Universal Robots PolyScope program: HeatPWF.urp

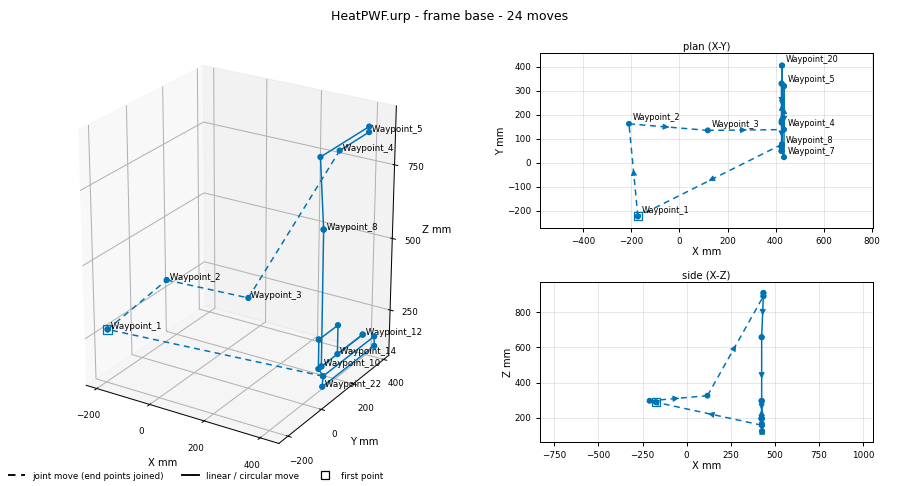
[picture p0: tool path of HeatPWF.urp in frame base, 24 of 24 moves have a stored position in this frame; points joined in program order, loops and branches not executed]
Program TDaiHeatPWF1 (installation=default directory=/programs/usbdisk_0/UR_URPs createdIn=5.11.0.108249 lastSavedIn=5.11.0.108249 robotSerialNumber=20215590035)
Calibrated DH parameters: a=[0.00016, -0.349388, -0.392209, -0.000059, 0.000026, 0]; d=[0.162575, -215.770964, 216.209801, -0.305241, 0.099656, 0.099253]; alpha=[1.570834, -0.001122, 0.007322, 1.56929, -1.570073, 0]; deltaTheta=[0, 0.606034, 5.685341, -0.008192, 0.000001, 0]
Robot Program (runOnlyOnce=true)
  MoveJ speed 60 deg/s, acceleration 80 deg/s^2 (useActiveTCP=true) feature=Base
    Waypoint Waypoint_1: TCP in base x=-173.333 y=-223.371 z=288.487 mm, rx=-2.2066 ry=-2.2292 rz=0.0202 rad; joints [-99.337, -57.321, -138.717, -73.565, 89.803, 80.13] deg; TCP offset x=0 y=0 z=26 mm, rx=0 ry=0 rz=0 rad
  MoveJ speed 60 deg/s, acceleration 80 deg/s^2 (useActiveTCP=true) feature=Base
    Waypoint Waypoint_2: TCP in base x=-210.394 y=161.858 z=296.687 mm, rx=-3.1305 ry=-0.0742 rz=0.0332 rad; joints [-187.188, -52.739, -139.358, -76.659, 90.078, 80.121] deg
  MoveJ speed 60 deg/s, acceleration 80 deg/s^2 (useActiveTCP=true) feature=Base
    Waypoint Waypoint_3: TCP in base x=117.831 y=134.656 z=325.784 mm, rx=-3.1162 ry=-0.0095 rz=0.0014 rad; joints [-262.681, -29.685, -139.379, -99.527, 90.347, 6.803] deg
  URCap Gripper Activate (Robotiq_Grippers, Robotiq Inc.) dataModel(ResetAndActivateKey=false)
  URCap Gripper (Robotiq_Grippers, Robotiq Inc.) dataModel(position=0.0, force=99.6078431372549, speed=99.6078431372549, positionInDouble=0.0, forceInDouble=99.6078431372549, speedInDouble=99.6078431372549, slaveIds=[9], blocking=true)
  MoveJ speed 60 deg/s, acceleration 80 deg/s^2 (useActiveTCP=true) feature=Base
    Waypoint Waypoint_4: TCP in base x=435.252 y=137.856 z=890.1 mm, rx=-1.5865 ry=-0.0166 rz=0.0088 rad; joints [-340.703, -101.32, -45.922, -34.906, 161.789, -2.225] deg; TCP offset x=0 y=0 z=26 mm, rx=0 ry=0 rz=0 rad
  MoveL speed 250 mm/s, acceleration 1200 mm/s^2 (useActiveTCP=true) feature=Base
    Waypoint Waypoint_5: TCP in base x=435.245 y=318.777 z=890.1 mm, rx=-1.5865 ry=-0.0165 rz=0.0088 rad; joints [-320.019, -108.883, -35.784, -36.509, 141.12, -1.021] deg; TCP offset x=0 y=0 z=26 mm, rx=0 ry=0 rz=0 rad
  URCap Gripper (Robotiq_Grippers, Robotiq Inc.) dataModel(position=100.0, force=99.6078431372549, speed=99.6078431372549, positionInDouble=100.0, forceInDouble=99.6078431372549, speedInDouble=99.6078431372549, slaveIds=[9], blocking=true)
  Wait Sleep waitTime=2
  MoveL speed 250 mm/s, acceleration 1200 mm/s^2 (useActiveTCP=true) feature=Base
    Waypoint Waypoint_6: TCP in base x=435.267 y=318.768 z=908.15 mm, rx=-1.5866 ry=-0.0165 rz=0.0088 rad; joints [-320.014, -111.696, -28.292, -41.223, 141.139, -1.062] deg; TCP offset x=0 y=0 z=26 mm, rx=0 ry=0 rz=0 rad
  MoveL speed 250 mm/s, acceleration 1200 mm/s^2 (useActiveTCP=true) feature=Base
    Waypoint Waypoint_7: TCP in base x=435.286 y=22.701 z=908.15 mm, rx=-1.5865 ry=-0.0165 rz=0.0088 rad; joints [-356.011, -102.521, -40.708, -50.091, 177.072, -13.563] deg; TCP offset x=0 y=0 z=26 mm, rx=0 ry=0 rz=0 rad
  MoveL speed 250 mm/s, acceleration 1200 mm/s^2 (useActiveTCP=true) feature=Base
    Waypoint Waypoint_8: TCP in base x=425.177 y=66.884 z=657.108 mm, rx=-1.5865 ry=-0.0165 rz=0.0088 rad; joints [-349.879, -91.671, -92.555, 0.602, 170.706, -3.792] deg; TCP offset x=0 y=0 z=26 mm, rx=0 ry=0 rz=0 rad
  MoveL speed 250 mm/s, acceleration 1200 mm/s^2 (useActiveTCP=true) feature=Base
    Waypoint Waypoint_9: TCP in base x=425.174 y=66.915 z=657.116 mm, rx=-0.9211 ry=1.6035 rz=-1.5828 rad; joints [-314.913, -78.501, -104.473, -2.311, 14.379, 4.931] deg
  MoveL speed 250 mm/s, acceleration 1200 mm/s^2 (useActiveTCP=true) feature=Base
    Waypoint Waypoint_10: TCP in base x=425.173 y=66.895 z=195.921 mm, rx=-0.9209 ry=1.6035 rz=-1.5828 rad; joints [-314.755, -129.845, -134.905, 80.997, 13.77, 3.359] deg
  MoveL speed 250 mm/s, acceleration 1200 mm/s^2 (useActiveTCP=true) feature=Base
    Waypoint Waypoint_11: TCP in base x=425.167 y=66.901 z=195.933 mm, rx=-0.0033 ry=-2.2326 rz=2.1976 rad; joints [-319.08, -111.028, -111.002, -136.209, 41.723, 178.135] deg
  MoveL speed 250 mm/s, acceleration 1200 mm/s^2 (useActiveTCP=true) feature=Base
    Waypoint Waypoint_12: TCP in base x=425.17 y=329.294 z=195.907 mm, rx=-0.0034 ry=-2.2325 rz=2.1977 rad; joints [-300.748, -128.821, -81.346, -148.586, 59.984, 178.716] deg
  MoveL speed 250 mm/s, acceleration 1200 mm/s^2 (useActiveTCP=true) feature=Base
    Waypoint Waypoint_13: TCP in base x=425.159 y=329.331 z=195.903 mm, rx=-1.222 ry=-1.2156 rz=1.1908 rad; joints [-317.144, -131.095, -77.257, -150.887, 133.697, 179.925] deg
  MoveL speed 250 mm/s, acceleration 1200 mm/s^2 (useActiveTCP=true) feature=Base
    Waypoint Waypoint_14: TCP in base x=425.186 y=166.978 z=195.927 mm, rx=-1.2221 ry=-1.2155 rz=1.1907 rad; joints [-329.777, -123.254, -91.096, -144.902, 121.111, 179.738] deg
  MoveL speed 250 mm/s, acceleration 1200 mm/s^2 (useActiveTCP=true) feature=Base
    Waypoint Waypoint_15: TCP in base x=425.176 y=166.963 z=296.274 mm, rx=-1.2221 ry=-1.2155 rz=1.1908 rad; joints [-329.771, -116.934, -84.699, -157.655, 121.031, 179.678] deg
  MoveL speed 250 mm/s, acceleration 1200 mm/s^2 (useActiveTCP=true) feature=Base
    Waypoint Waypoint_16: TCP in base x=425.176 y=48.726 z=296.245 mm, rx=-1.2221 ry=-1.2155 rz=1.1908 rad; joints [-341.038, -114.052, -89.038, -156.17, 109.773, 179.522] deg
  MoveL speed 250 mm/s, acceleration 1200 mm/s^2 (useActiveTCP=true) feature=Base
    Waypoint Waypoint_17: TCP in base x=425.169 y=48.71 z=296.237 mm, rx=-1.572 ry=-0.2489 rz=0.2377 rad; joints [-352.046, -103.026, -104.27, -150.378, 170.47, 181.942] deg
  MoveL speed 250 mm/s, acceleration 1200 mm/s^2 (useActiveTCP=true) feature=Base
    Waypoint Waypoint_18: TCP in base x=425.17 y=48.7 z=195.307 mm, rx=-1.572 ry=-0.2488 rz=0.2376 rad; joints [-352.06, -111.045, -111.113, -135.079, 170.549, 182.387] deg
  MoveJ speed 60 deg/s, acceleration 80 deg/s^2 (useActiveTCP=true) feature=Base
    Waypoint Waypoint_19: TCP in base x=426.358 y=76.543 z=158.403 mm, rx=-1.5462 ry=-0.0196 rz=0.0152 rad; joints [-348.42, -110.597, -121.041, -118.722, 190.825, 189.361] deg
  MoveL speed 250 mm/s, acceleration 1200 mm/s^2 (useActiveTCP=true) feature=Base
    Waypoint Waypoint_20: TCP in base x=426.365 y=404.622 z=158.318 mm, rx=-1.5463 ry=-0.0195 rz=0.0151 rad; joints [-311.781, -119.872, -105.068, -132.746, 227.334, 181.68] deg
  MoveL speed 250 mm/s, acceleration 1200 mm/s^2 (useActiveTCP=true) feature=Base
    Waypoint Waypoint_21: TCP in base x=427.366 y=404.665 z=124.443 mm, rx=-1.5462 ry=-0.0196 rz=0.0151 rad; joints [-311.87, -123.421, -105.813, -128.466, 227.261, 181.646] deg
  Wait Sleep waitTime=1
  URCap Gripper (Robotiq_Grippers, Robotiq Inc.) dataModel(position=0.0, force=0.0, speed=0.0, positionInDouble=0.0, forceInDouble=0.0, speedInDouble=0.0, slaveIds=[9], blocking=true)
  Wait Sleep waitTime=2
  MoveL speed 250 mm/s, acceleration 1200 mm/s^2 (useActiveTCP=true) feature=Base
    Waypoint Waypoint_22: TCP in base x=427.404 y=70.563 z=124.489 mm, rx=-1.5461 ry=-0.0197 rz=0.015 rad; joints [-349.275, -115.036, -121.922, -112.808, 190.002, 189.948] deg
  MoveL speed 250 mm/s, acceleration 1200 mm/s^2 (useActiveTCP=true) feature=Base
    Waypoint Waypoint_19: TCP in base x=426.358 y=76.543 z=158.403 mm, rx=-1.5462 ry=-0.0196 rz=0.0152 rad; joints [-348.42, -110.597, -121.041, -118.722, 190.825, 189.361] deg
  MoveJ speed 60 deg/s, acceleration 80 deg/s^2 (useActiveTCP=true) feature=Base
    Waypoint Waypoint_1: TCP in base x=-173.333 y=-223.371 z=288.487 mm, rx=-2.2066 ry=-2.2292 rz=0.0202 rad; joints [-99.337, -57.321, -138.717, -73.565, 89.803, 80.13] deg
  URCap Gripper (Robotiq_Grippers, Robotiq Inc.) dataModel(position=100.0, force=0.0, speed=0.0, positionInDouble=100.0, forceInDouble=0.0, speedInDouble=0.0, slaveIds=[9], blocking=true)
